FUNCTION CreateDTL : DTL

CreateDTL.YEAR		:= 0;
CreateDTL.MONTH		:= 0;
CreateDTL.DAY			:= 0;
CreateDTL.HOUR		:= 0;
CreateDTL.MINUTE		:= 0;
CreateDTL.SECOND		:= 0;
CreateDTL.MILLISECOND	:= 0;

END_FUNCTION

(* stored: Version 1.1.0.1, ProductVersion 3.1.4026.4
   POU CreateDTL: Id {09c3a8fc-7199-4dc5-bad7-159cec065828}, SpecialFunc None *)
